INTERFACE I_TestEventHandler EXTENDS I_EventHandlerBase

METHOD OnCustomEvent
VAR_INPUT
    EventArgs : I_StreamReader;
END_VAR
END_METHOD

END_INTERFACE

(* stored: Version 1.1.0.1, ProductVersion 3.1.4024.4
   Itf I_TestEventHandler: Id {5c9f4999-f01f-4959-839d-129089c37d61}
   Method OnCustomEvent: Id {83d06d90-640d-490c-a78c-3e28192ff3d4} *)
